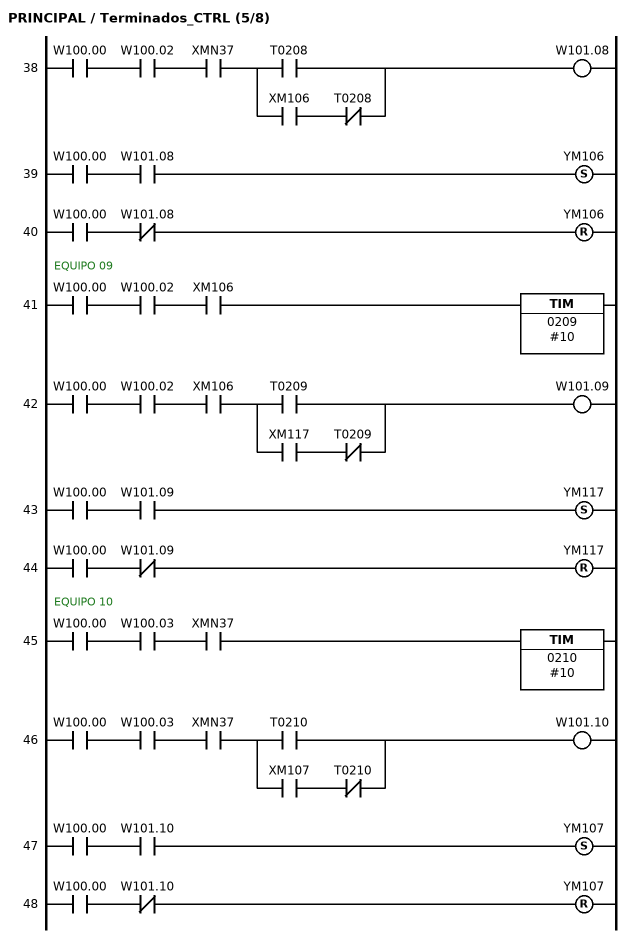
; [picture p24: PRINCIPAL / Terminados_CTRL, rungs 38-48]
; rung 38
LD W100.00
AND W100.02
AND XMN37
LD T0208
LD XM106
ANDNOT T0208
ORLD
ANDLD
OUT W101.08
; rung 39
LD W100.00
AND W101.08
SET YM106
; rung 40
LD W100.00
ANDNOT W101.08
RSET YM106
; rung 41: EQUIPO 09
LD W100.00
AND W100.02
AND XM106
TIM 0209 #10
; rung 42
LD W100.00
AND W100.02
AND XM106
LD T0209
LD XM117
ANDNOT T0209
ORLD
ANDLD
OUT W101.09
; rung 43
LD W100.00
AND W101.09
SET YM117
; rung 44
LD W100.00
ANDNOT W101.09
RSET YM117
; rung 45: EQUIPO 10
LD W100.00
AND W100.03
AND XMN37
TIM 0210 #10
; rung 46
LD W100.00
AND W100.03
AND XMN37
LD T0210
LD XM107
ANDNOT T0210
ORLD
ANDLD
OUT W101.10
; rung 47
LD W100.00
AND W101.10
SET YM107
; rung 48
LD W100.00
ANDNOT W101.10
RSET YM107

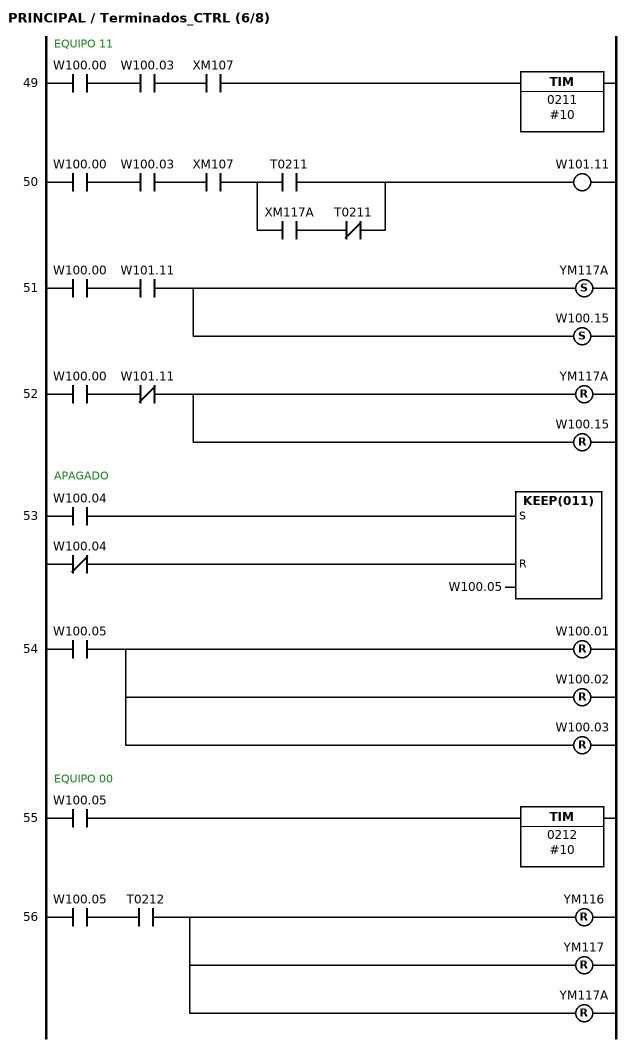
; rung 49: EQUIPO 11
LD W100.00
AND W100.03
AND XM107
TIM 0211 #10
; rung 50
LD W100.00
AND W100.03
AND XM107
LD T0211
LD XM117A
ANDNOT T0211
ORLD
ANDLD
OUT W101.11
; rung 51
LD W100.00
AND W101.11
SET YM117A
SET W100.15
; rung 52
LD W100.00
ANDNOT W101.11
RSET YM117A
RSET W100.15
; rung 53: APAGADO
LD W100.04
LDNOT W100.04
KEEP(011) W100.05
; rung 54
LD W100.05
RSET W100.01
RSET W100.02
RSET W100.03
; rung 55: EQUIPO 00
LD W100.05
TIM 0212 #10
; rung 56
LD W100.05
AND T0212
RSET YM116
RSET YM117
RSET YM117A

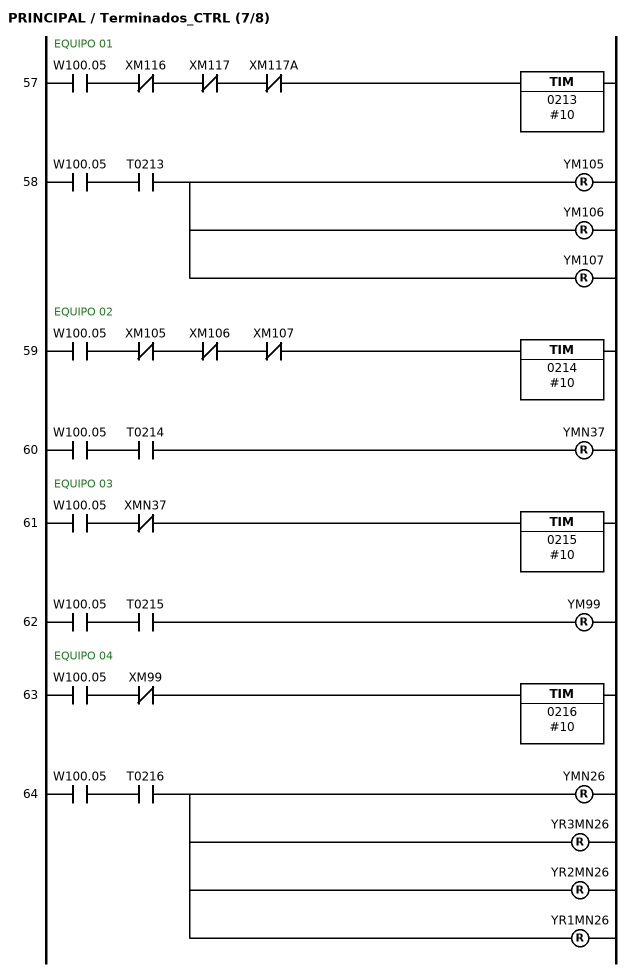
; rung 57: EQUIPO 01
LD W100.05
ANDNOT XM116
ANDNOT XM117
ANDNOT XM117A
TIM 0213 #10
; rung 58
LD W100.05
AND T0213
RSET YM105
RSET YM106
RSET YM107
; rung 59: EQUIPO 02
LD W100.05
ANDNOT XM105
ANDNOT XM106
ANDNOT XM107
TIM 0214 #10
; rung 60
LD W100.05
AND T0214
RSET YMN37
; rung 61: EQUIPO 03
LD W100.05
ANDNOT XMN37
TIM 0215 #10
; rung 62
LD W100.05
AND T0215
RSET YM99
; rung 63: EQUIPO 04
LD W100.05
ANDNOT XM99
TIM 0216 #10
; rung 64
LD W100.05
AND T0216
RSET YMN26
RSET YR3MN26
RSET YR2MN26
RSET YR1MN26

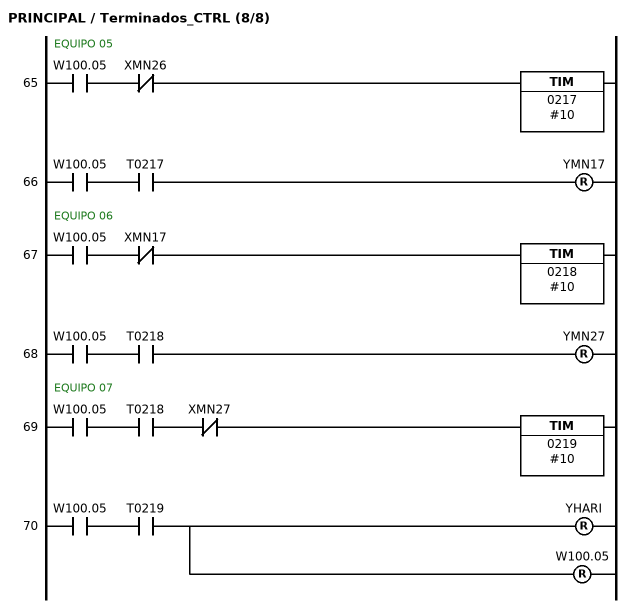
; rung 65: EQUIPO 05
LD W100.05
ANDNOT XMN26
TIM 0217 #10
; rung 66
LD W100.05
AND T0217
RSET YMN17
; rung 67: EQUIPO 06
LD W100.05
ANDNOT XMN17
TIM 0218 #10
; rung 68
LD W100.05
AND T0218
RSET YMN27
; rung 69: EQUIPO 07
LD W100.05
AND T0218
ANDNOT XMN27
TIM 0219 #10
; rung 70
LD W100.05
AND T0219
RSET YHARI
RSET W100.05

### Section Terminados_OUT

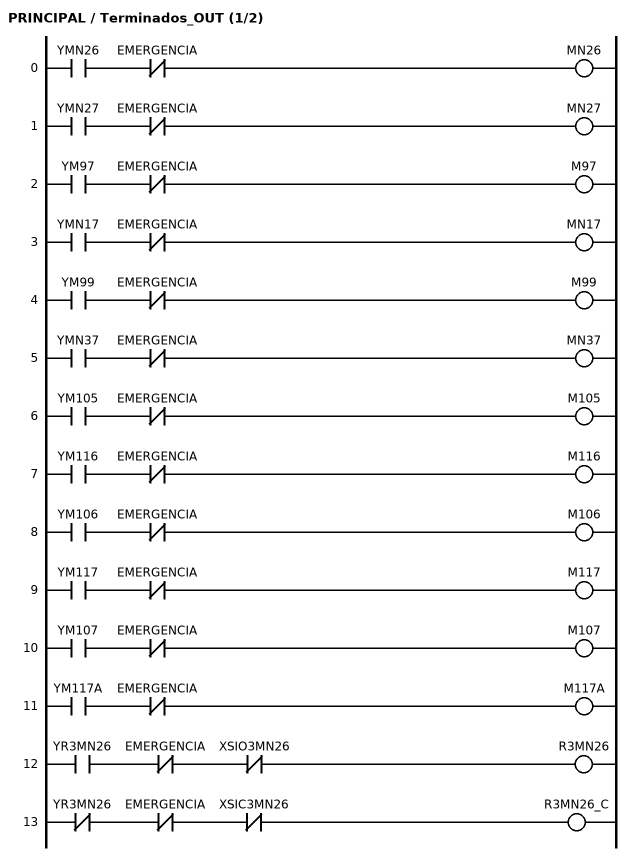
; rung 0
LD YMN26
ANDNOT EMERGENCIA
OUT MN26
; rung 1
LD YMN27
ANDNOT EMERGENCIA
OUT MN27
; rung 2
LD YM97
ANDNOT EMERGENCIA
OUT M97
; rung 3
LD YMN17
ANDNOT EMERGENCIA
OUT MN17
; rung 4
LD YM99
ANDNOT EMERGENCIA
OUT M99
; rung 5
LD YMN37
ANDNOT EMERGENCIA
OUT MN37
; rung 6
LD YM105
ANDNOT EMERGENCIA
OUT M105
; rung 7
LD YM116
ANDNOT EMERGENCIA
OUT M116
; rung 8
LD YM106
ANDNOT EMERGENCIA
OUT M106
; rung 9
LD YM117
ANDNOT EMERGENCIA
OUT M117
; rung 10
LD YM107
ANDNOT EMERGENCIA
OUT M107
; rung 11
LD YM117A
ANDNOT EMERGENCIA
OUT M117A
; rung 12
LD YR3MN26
ANDNOT EMERGENCIA
ANDNOT XSIO3MN26
OUT R3MN26
; rung 13
LDNOT YR3MN26
ANDNOT EMERGENCIA
ANDNOT XSIC3MN26
OUT R3MN26_C

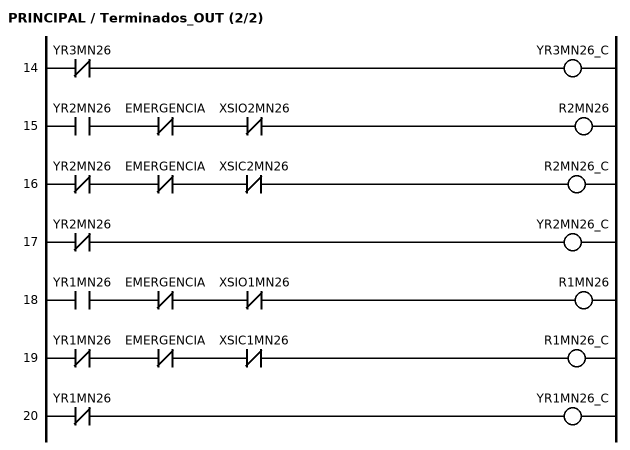
; rung 14
LDNOT YR3MN26
OUT YR3MN26_C
; rung 15
LD YR2MN26
ANDNOT EMERGENCIA
ANDNOT XSIO2MN26
OUT R2MN26
; rung 16
LDNOT YR2MN26
ANDNOT EMERGENCIA
ANDNOT XSIC2MN26
OUT R2MN26_C
; rung 17
LDNOT YR2MN26
OUT YR2MN26_C
; rung 18
LD YR1MN26
ANDNOT EMERGENCIA
ANDNOT XSIO1MN26
OUT R1MN26
; rung 19
LDNOT YR1MN26
ANDNOT EMERGENCIA
ANDNOT XSIC1MN26
OUT R1MN26_C
; rung 20
LDNOT YR1MN26
OUT YR1MN26_C

### Section LPZ_T1_v1_CTRL

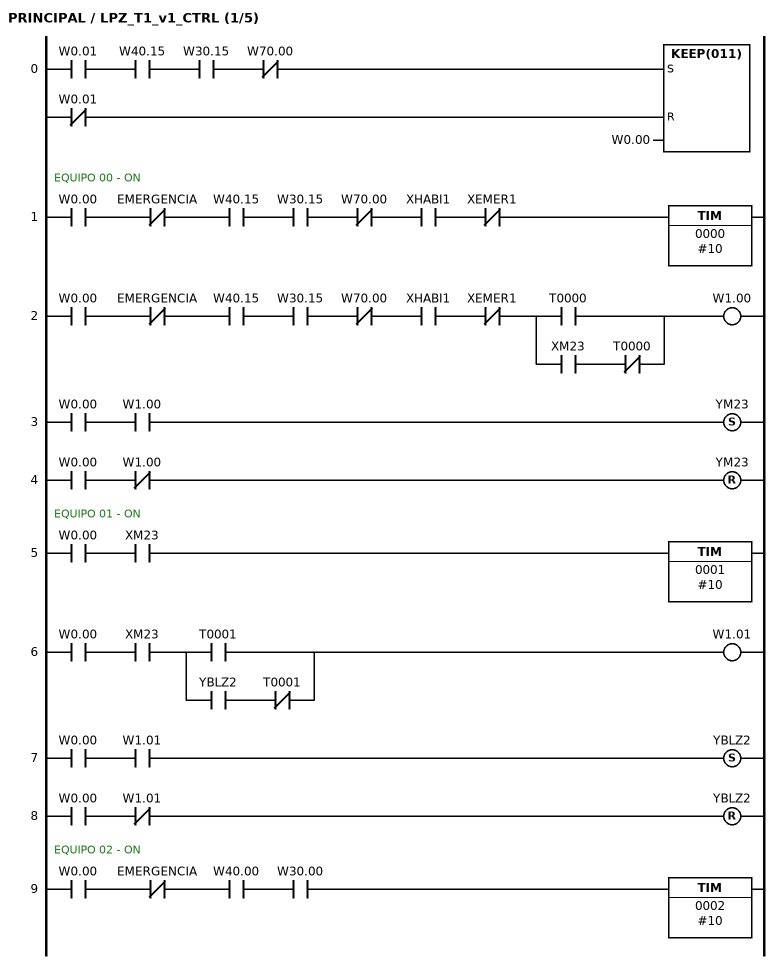
; rung 0
LD W0.01
AND W40.15
AND W30.15
ANDNOT W70.00
LDNOT W0.01
KEEP(011) W0.00
; rung 1: EQUIPO 00 - ON
LD W0.00
ANDNOT EMERGENCIA
AND W40.15
AND W30.15
ANDNOT W70.00
AND XHABI1
ANDNOT XEMER1
TIM 0000 #10
; rung 2
LD W0.00
ANDNOT EMERGENCIA
AND W40.15
AND W30.15
ANDNOT W70.00
AND XHABI1
ANDNOT XEMER1
LD T0000
LD XM23
ANDNOT T0000
ORLD
ANDLD
OUT W1.00
; rung 3
LD W0.00
AND W1.00
SET YM23
; rung 4
LD W0.00
ANDNOT W1.00
RSET YM23
; rung 5: EQUIPO 01 - ON
LD W0.00
AND XM23
TIM 0001 #10
; rung 6
LD W0.00
AND XM23
LD T0001
LD YBLZ2
ANDNOT T0001
ORLD
ANDLD
OUT W1.01
; rung 7
LD W0.00
AND W1.01
SET YBLZ2
; rung 8
LD W0.00
ANDNOT W1.01
RSET YBLZ2
; rung 9: EQUIPO 02 - ON
LD W0.00
ANDNOT EMERGENCIA
AND W40.00
AND W30.00
TIM 0002 #10

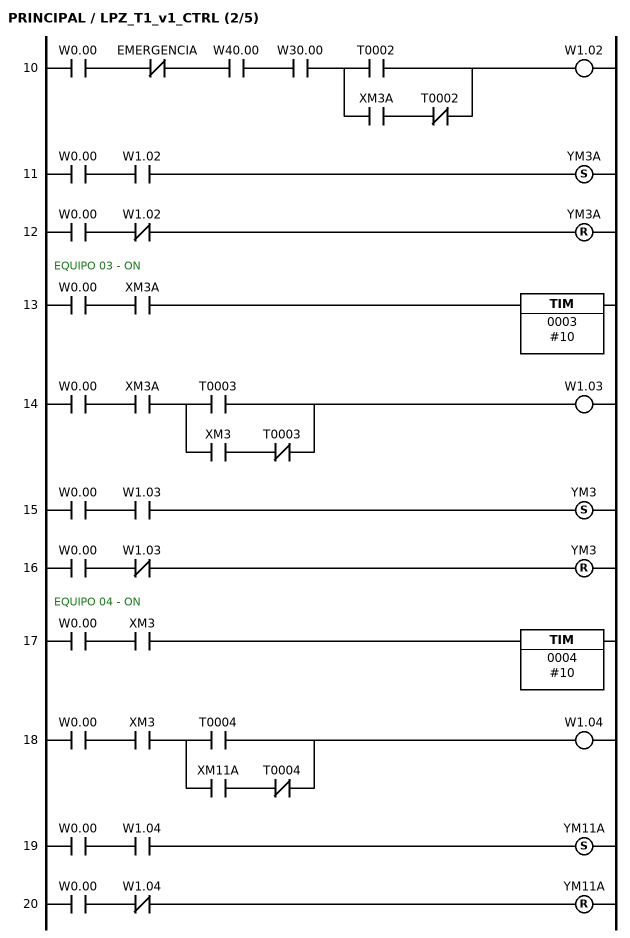
; rung 10
LD W0.00
ANDNOT EMERGENCIA
AND W40.00
AND W30.00
LD T0002
LD XM3A
ANDNOT T0002
ORLD
ANDLD
OUT W1.02
; rung 11
LD W0.00
AND W1.02
SET YM3A
; rung 12
LD W0.00
ANDNOT W1.02
RSET YM3A
; rung 13: EQUIPO 03 - ON
LD W0.00
AND XM3A
TIM 0003 #10
; rung 14
LD W0.00
AND XM3A
LD T0003
LD XM3
ANDNOT T0003
ORLD
ANDLD
OUT W1.03
; rung 15
LD W0.00
AND W1.03
SET YM3
; rung 16
LD W0.00
ANDNOT W1.03
RSET YM3
; rung 17: EQUIPO 04 - ON
LD W0.00
AND XM3
TIM 0004 #10
; rung 18
LD W0.00
AND XM3
LD T0004
LD XM11A
ANDNOT T0004
ORLD
ANDLD
OUT W1.04
; rung 19
LD W0.00
AND W1.04
SET YM11A
; rung 20
LD W0.00
ANDNOT W1.04
RSET YM11A

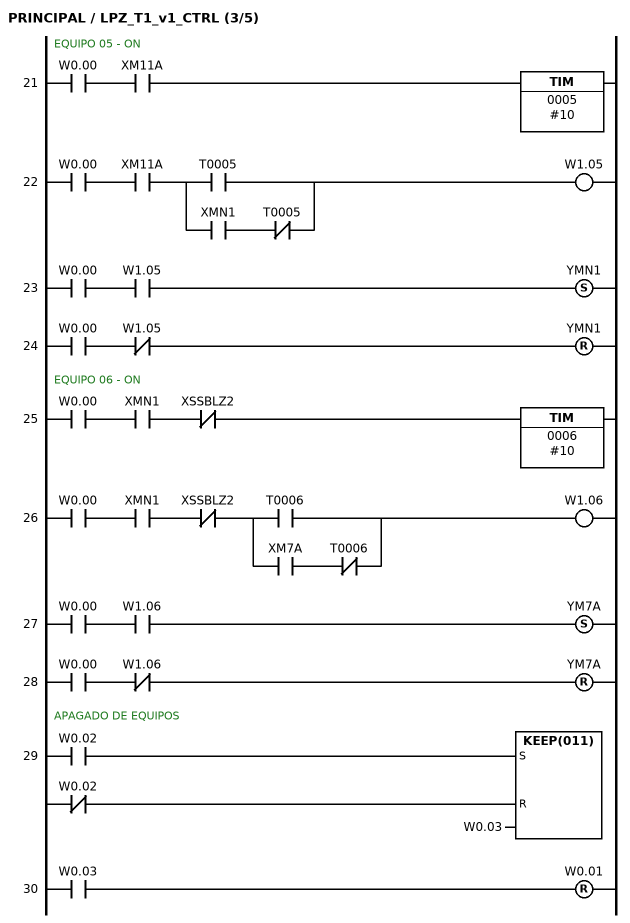
; rung 21: EQUIPO 05 - ON
LD W0.00
AND XM11A
TIM 0005 #10
; rung 22
LD W0.00
AND XM11A
LD T0005
LD XMN1
ANDNOT T0005
ORLD
ANDLD
OUT W1.05
; rung 23
LD W0.00
AND W1.05
SET YMN1
; rung 24
LD W0.00
ANDNOT W1.05
RSET YMN1
; rung 25: EQUIPO 06 - ON
LD W0.00
AND XMN1
ANDNOT XSSBLZ2
TIM 0006 #10
; rung 26
LD W0.00
AND XMN1
ANDNOT XSSBLZ2
LD T0006
LD XM7A
ANDNOT T0006
ORLD
ANDLD
OUT W1.06
; rung 27
LD W0.00
AND W1.06
SET YM7A
; rung 28
LD W0.00
ANDNOT W1.06
RSET YM7A
; rung 29: APAGADO DE EQUIPOS
LD W0.02
LDNOT W0.02
KEEP(011) W0.03
; rung 30
LD W0.03
RSET W0.01

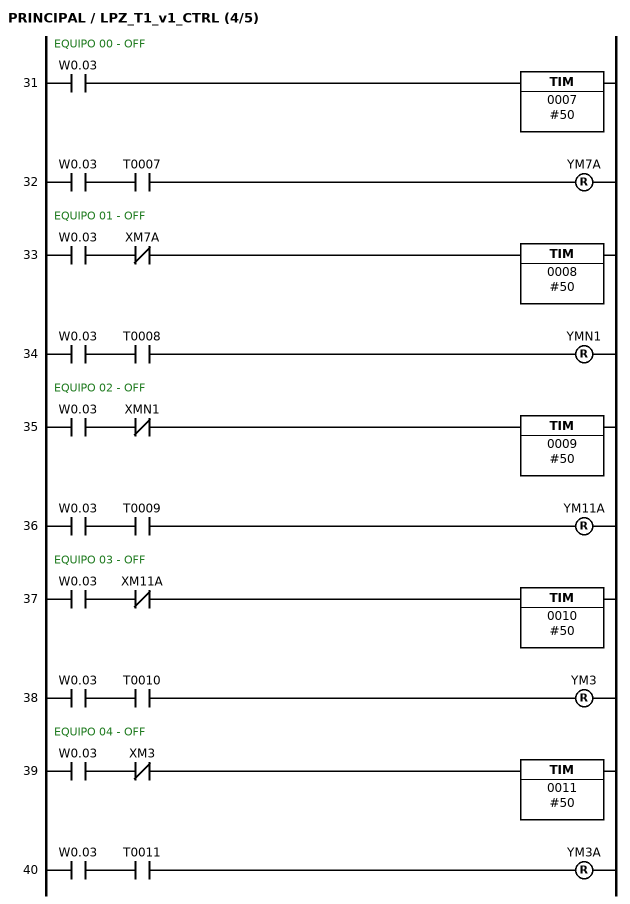
; rung 31: EQUIPO 00 - OFF
LD W0.03
TIM 0007 #50
; rung 32
LD W0.03
AND T0007
RSET YM7A
; rung 33: EQUIPO 01 - OFF
LD W0.03
ANDNOT XM7A
TIM 0008 #50
; rung 34
LD W0.03
AND T0008
RSET YMN1
; rung 35: EQUIPO 02 - OFF
LD W0.03
ANDNOT XMN1
TIM 0009 #50
; rung 36
LD W0.03
AND T0009
RSET YM11A
; rung 37: EQUIPO 03 - OFF
LD W0.03
ANDNOT XM11A
TIM 0010 #50
; rung 38
LD W0.03
AND T0010
RSET YM3
; rung 39: EQUIPO 04 - OFF
LD W0.03
ANDNOT XM3
TIM 0011 #50
; rung 40
LD W0.03
AND T0011
RSET YM3A

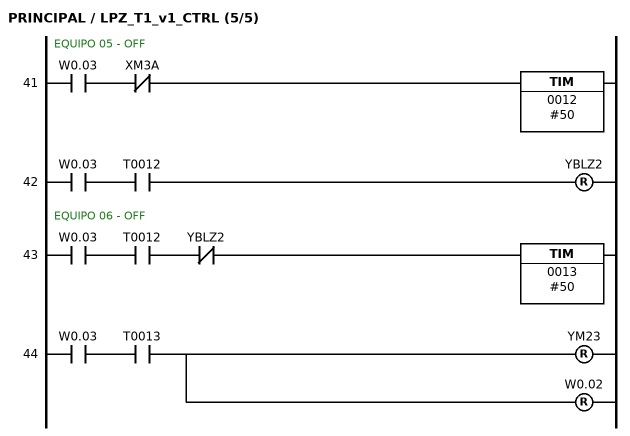
; rung 41: EQUIPO 05 - OFF
LD W0.03
ANDNOT XM3A
TIM 0012 #50
; rung 42
LD W0.03
AND T0012
RSET YBLZ2
; rung 43: EQUIPO 06 - OFF
LD W0.03
AND T0012
ANDNOT YBLZ2
TIM 0013 #50
; rung 44
LD W0.03
AND T0013
RSET YM23
RSET W0.02

### Section LPZ_T1_v2_CTRL

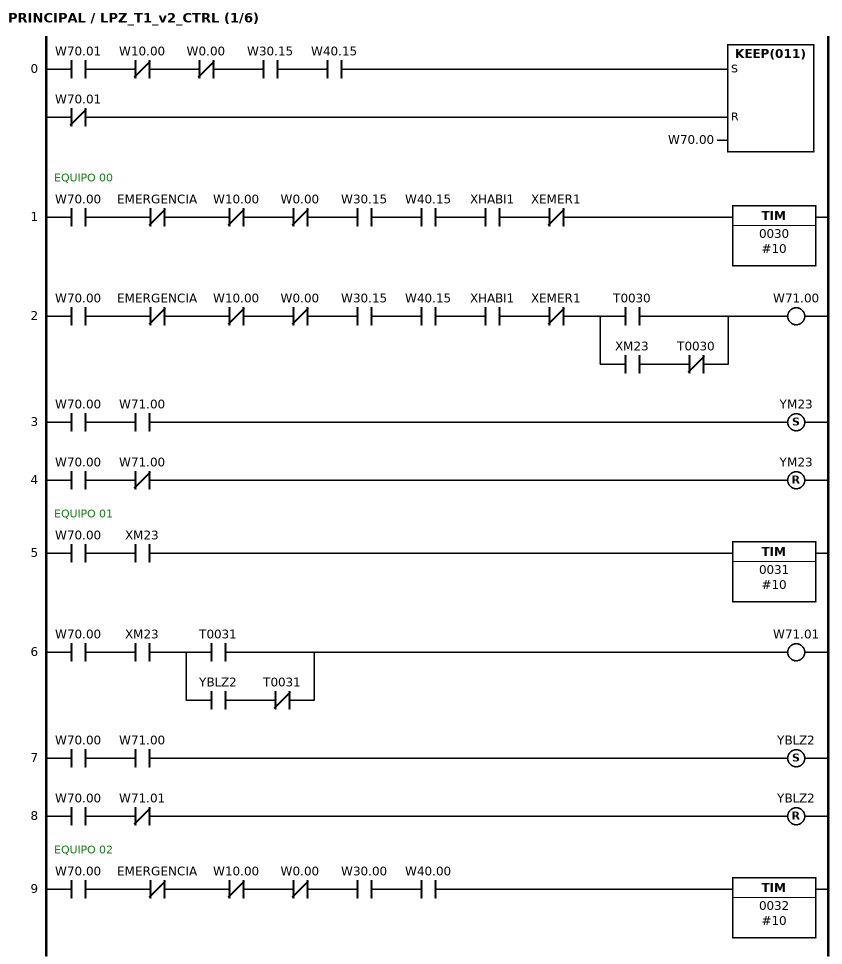
; rung 0
LD W70.01
ANDNOT W10.00
ANDNOT W0.00
AND W30.15
AND W40.15
LDNOT W70.01
KEEP(011) W70.00
; rung 1: EQUIPO 00
LD W70.00
ANDNOT EMERGENCIA
ANDNOT W10.00
ANDNOT W0.00
AND W30.15
AND W40.15
AND XHABI1
ANDNOT XEMER1
TIM 0030 #10
; rung 2
LD W70.00
ANDNOT EMERGENCIA
ANDNOT W10.00
ANDNOT W0.00
AND W30.15
AND W40.15
AND XHABI1
ANDNOT XEMER1
LD T0030
LD XM23
ANDNOT T0030
ORLD
ANDLD
OUT W71.00
; rung 3
LD W70.00
AND W71.00
SET YM23
; rung 4
LD W70.00
ANDNOT W71.00
RSET YM23
; rung 5: EQUIPO 01
LD W70.00
AND XM23
TIM 0031 #10
; rung 6
LD W70.00
AND XM23
LD T0031
LD YBLZ2
ANDNOT T0031
ORLD
ANDLD
OUT W71.01
; rung 7
LD W70.00
AND W71.00
SET YBLZ2
; rung 8
LD W70.00
ANDNOT W71.01
RSET YBLZ2
; rung 9: EQUIPO 02
LD W70.00
ANDNOT EMERGENCIA
ANDNOT W10.00
ANDNOT W0.00
AND W30.00
AND W40.00
TIM 0032 #10

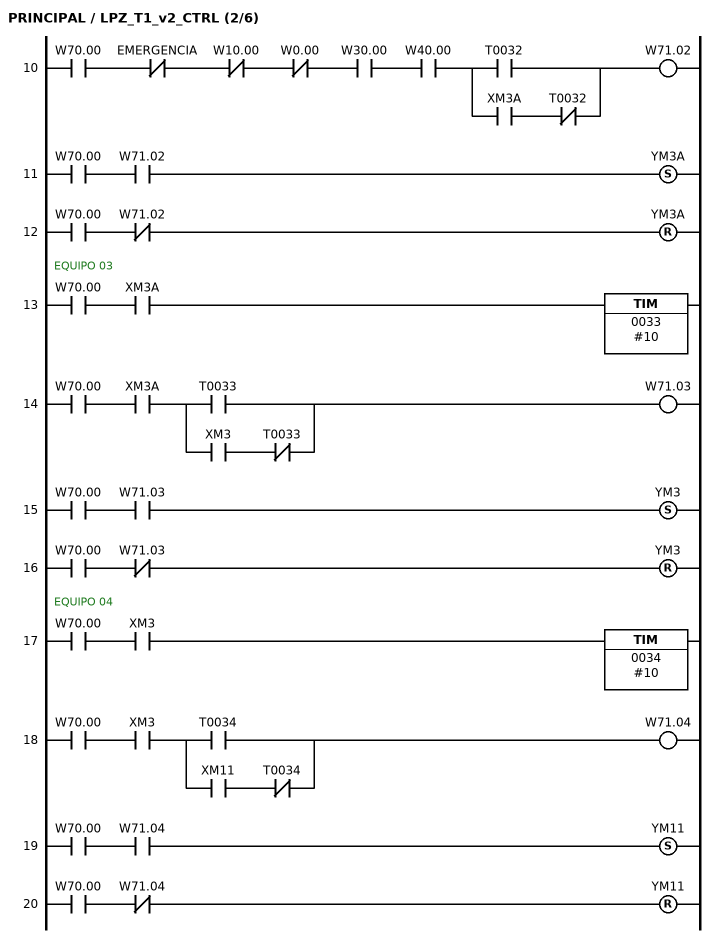
; rung 10
LD W70.00
ANDNOT EMERGENCIA
ANDNOT W10.00
ANDNOT W0.00
AND W30.00
AND W40.00
LD T0032
LD XM3A
ANDNOT T0032
ORLD
ANDLD
OUT W71.02
; rung 11
LD W70.00
AND W71.02
SET YM3A
; rung 12
LD W70.00
ANDNOT W71.02
RSET YM3A
; rung 13: EQUIPO 03
LD W70.00
AND XM3A
TIM 0033 #10
; rung 14
LD W70.00
AND XM3A
LD T0033
LD XM3
ANDNOT T0033
ORLD
ANDLD
OUT W71.03
; rung 15
LD W70.00
AND W71.03
SET YM3
; rung 16
LD W70.00
ANDNOT W71.03
RSET YM3
; rung 17: EQUIPO 04
LD W70.00
AND XM3
TIM 0034 #10
; rung 18
LD W70.00
AND XM3
LD T0034
LD XM11
ANDNOT T0034
ORLD
ANDLD
OUT W71.04
; rung 19
LD W70.00
AND W71.04
SET YM11
; rung 20
LD W70.00
ANDNOT W71.04
RSET YM11

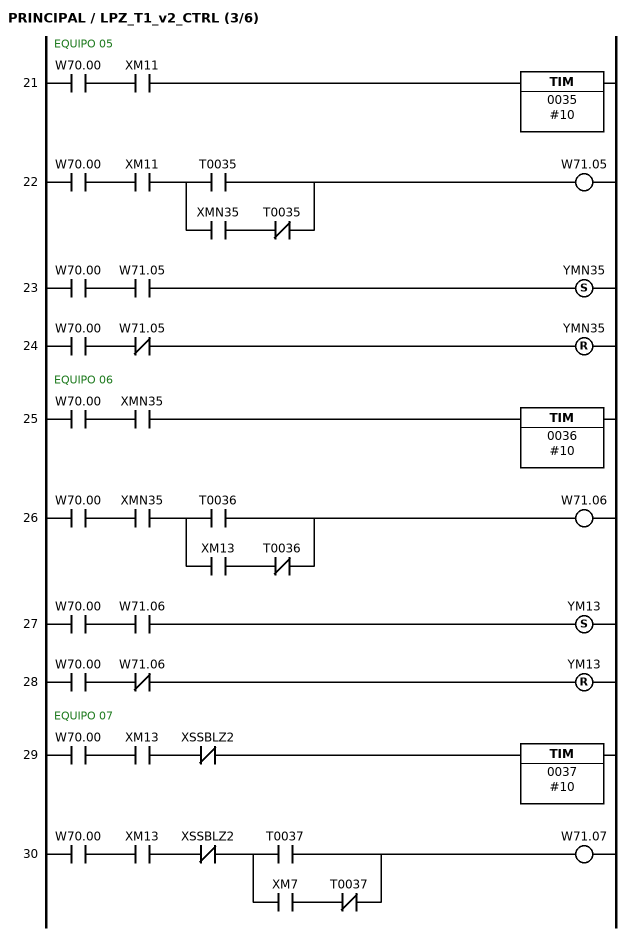
; rung 21: EQUIPO 05
LD W70.00
AND XM11
TIM 0035 #10
; rung 22
LD W70.00
AND XM11
LD T0035
LD XMN35
ANDNOT T0035
ORLD
ANDLD
OUT W71.05
; rung 23
LD W70.00
AND W71.05
SET YMN35
; rung 24
LD W70.00
ANDNOT W71.05
RSET YMN35
; rung 25: EQUIPO 06
LD W70.00
AND XMN35
TIM 0036 #10
; rung 26
LD W70.00
AND XMN35
LD T0036
LD XM13
ANDNOT T0036
ORLD
ANDLD
OUT W71.06
; rung 27
LD W70.00
AND W71.06
SET YM13
; rung 28
LD W70.00
ANDNOT W71.06
RSET YM13
; rung 29: EQUIPO 07
LD W70.00
AND XM13
ANDNOT XSSBLZ2
TIM 0037 #10
; rung 30
LD W70.00
AND XM13
ANDNOT XSSBLZ2
LD T0037
LD XM7
ANDNOT T0037
ORLD
ANDLD
OUT W71.07

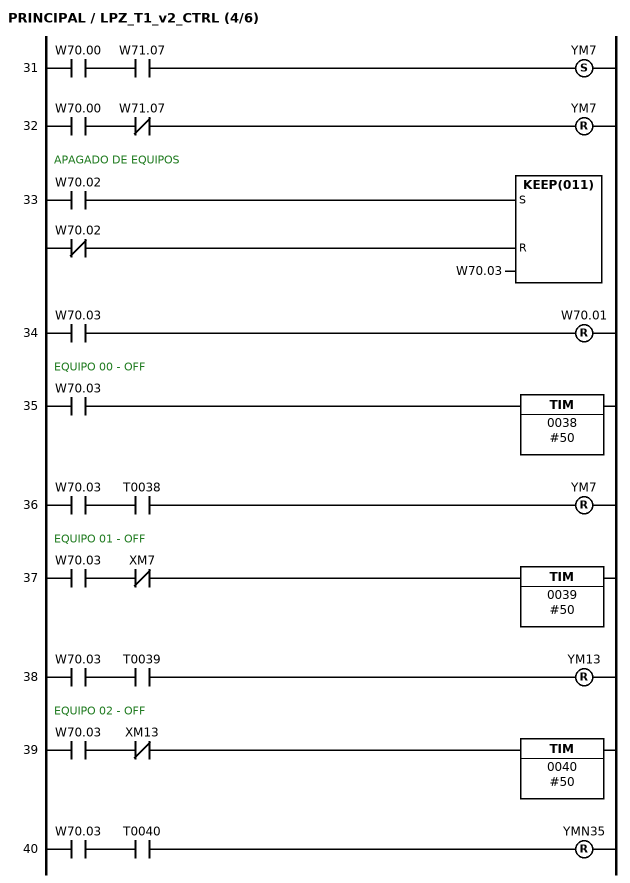
; rung 31
LD W70.00
AND W71.07
SET YM7
; rung 32
LD W70.00
ANDNOT W71.07
RSET YM7
; rung 33: APAGADO DE EQUIPOS
LD W70.02
LDNOT W70.02
KEEP(011) W70.03
; rung 34
LD W70.03
RSET W70.01
; rung 35: EQUIPO 00 - OFF
LD W70.03
TIM 0038 #50
; rung 36
LD W70.03
AND T0038
RSET YM7
; rung 37: EQUIPO 01 - OFF
LD W70.03
ANDNOT XM7
TIM 0039 #50
; rung 38
LD W70.03
AND T0039
RSET YM13
; rung 39: EQUIPO 02 - OFF
LD W70.03
ANDNOT XM13
TIM 0040 #50
; rung 40
LD W70.03
AND T0040
RSET YMN35

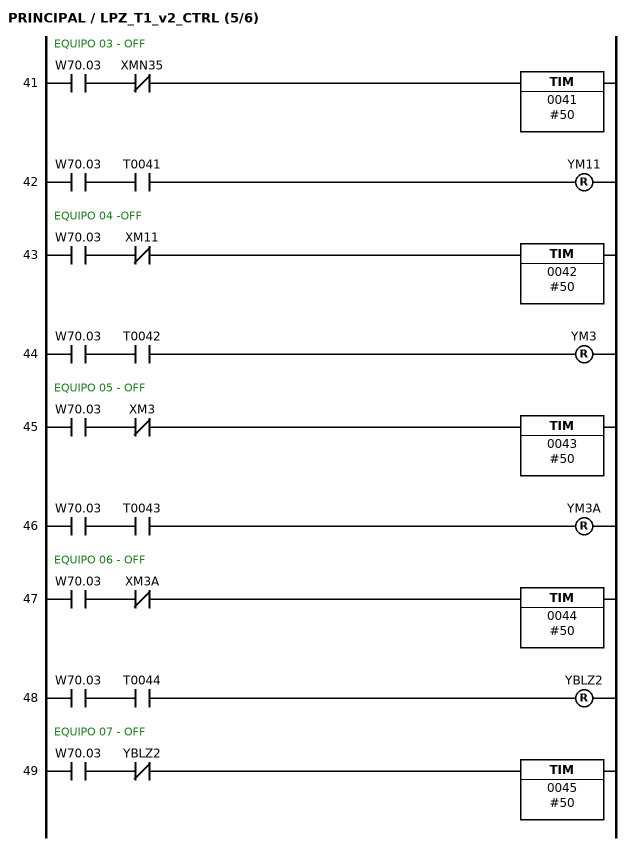
; rung 41: EQUIPO 03 - OFF
LD W70.03
ANDNOT XMN35
TIM 0041 #50
; rung 42
LD W70.03
AND T0041
RSET YM11
; rung 43: EQUIPO 04 -OFF
LD W70.03
ANDNOT XM11
TIM 0042 #50
; rung 44
LD W70.03
AND T0042
RSET YM3
; rung 45: EQUIPO 05 - OFF
LD W70.03
ANDNOT XM3
TIM 0043 #50
; rung 46
LD W70.03
AND T0043
RSET YM3A
; rung 47: EQUIPO 06 - OFF
LD W70.03
ANDNOT XM3A
TIM 0044 #50
; rung 48
LD W70.03
AND T0044
RSET YBLZ2
; rung 49: EQUIPO 07 - OFF
LD W70.03
ANDNOT YBLZ2
TIM 0045 #50

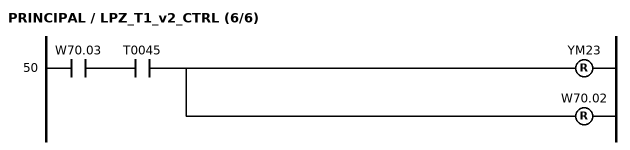
; rung 50
LD W70.03
AND T0045
RSET YM23
RSET W70.02

### Section LPZ_T1_OUT

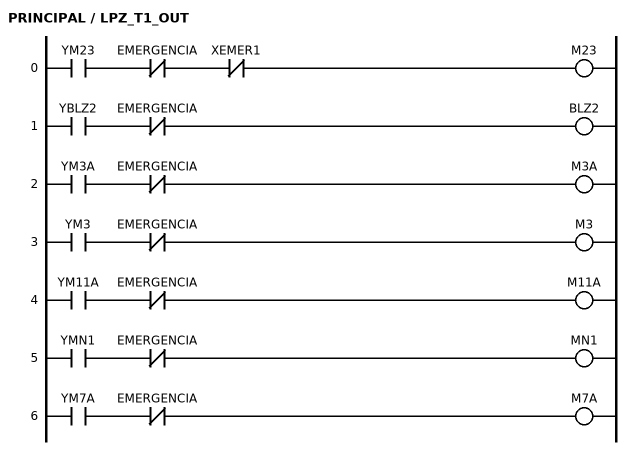
; rung 0
LD YM23
ANDNOT EMERGENCIA
ANDNOT XEMER1
OUT M23
; rung 1
LD YBLZ2
ANDNOT EMERGENCIA
OUT BLZ2
; rung 2
LD YM3A
ANDNOT EMERGENCIA
OUT M3A
; rung 3
LD YM3
ANDNOT EMERGENCIA
OUT M3
; rung 4
LD YM11A
ANDNOT EMERGENCIA
OUT M11A
; rung 5
LD YMN1
ANDNOT EMERGENCIA
OUT MN1
; rung 6
LD YM7A
ANDNOT EMERGENCIA
OUT M7A

### Section LPZ_2Rociado_CTRL

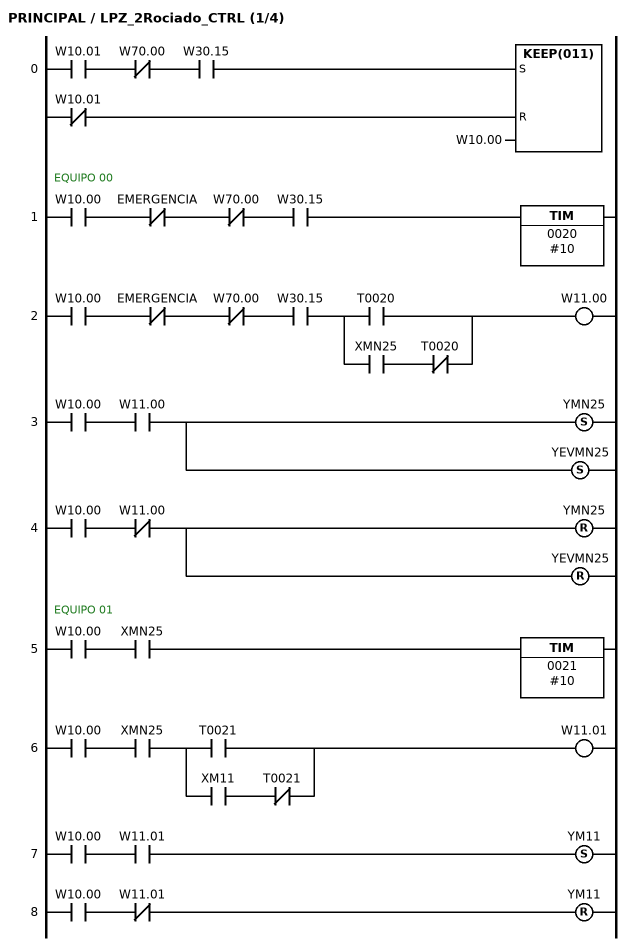
; rung 0
LD W10.01
ANDNOT W70.00
AND W30.15
LDNOT W10.01
KEEP(011) W10.00
; rung 1: EQUIPO 00
LD W10.00
ANDNOT EMERGENCIA
ANDNOT W70.00
AND W30.15
TIM 0020 #10
; rung 2
LD W10.00
ANDNOT EMERGENCIA
ANDNOT W70.00
AND W30.15
LD T0020
LD XMN25
ANDNOT T0020
ORLD
ANDLD
OUT W11.00
; rung 3
LD W10.00
AND W11.00
SET YMN25
SET YEVMN25
; rung 4
LD W10.00
ANDNOT W11.00
RSET YMN25
RSET YEVMN25
; rung 5: EQUIPO 01
LD W10.00
AND XMN25
TIM 0021 #10
; rung 6
LD W10.00
AND XMN25
LD T0021
LD XM11
ANDNOT T0021
ORLD
ANDLD
OUT W11.01
; rung 7
LD W10.00
AND W11.01
SET YM11
; rung 8
LD W10.00
ANDNOT W11.01
RSET YM11

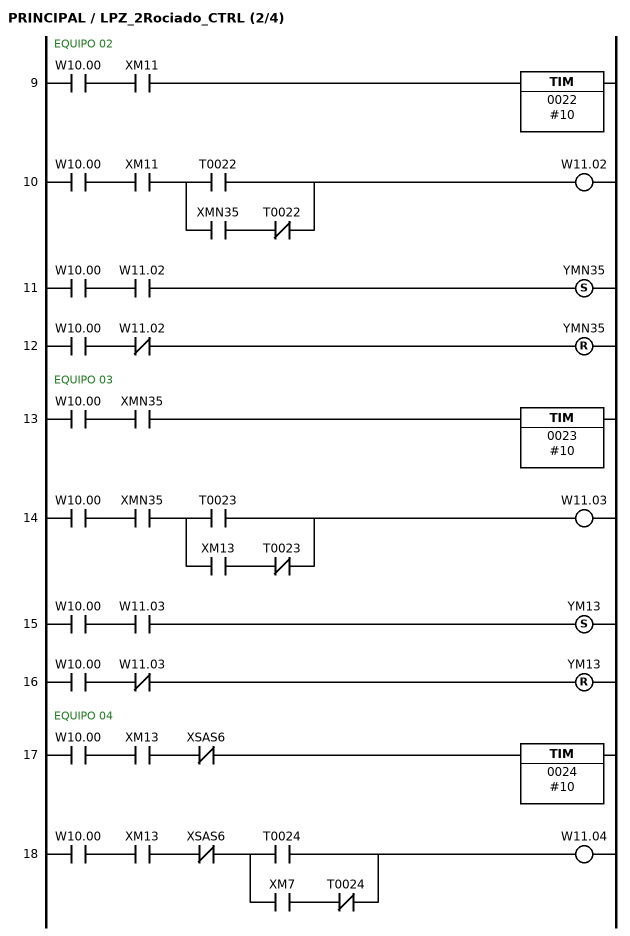
; rung 9: EQUIPO 02
LD W10.00
AND XM11
TIM 0022 #10
; rung 10
LD W10.00
AND XM11
LD T0022
LD XMN35
ANDNOT T0022
ORLD
ANDLD
OUT W11.02
; rung 11
LD W10.00
AND W11.02
SET YMN35
; rung 12
LD W10.00
ANDNOT W11.02
RSET YMN35
; rung 13: EQUIPO 03
LD W10.00
AND XMN35
TIM 0023 #10
; rung 14
LD W10.00
AND XMN35
LD T0023
LD XM13
ANDNOT T0023
ORLD
ANDLD
OUT W11.03
; rung 15
LD W10.00
AND W11.03
SET YM13
; rung 16
LD W10.00
ANDNOT W11.03
RSET YM13
; rung 17: EQUIPO 04
LD W10.00
AND XM13
ANDNOT XSAS6
TIM 0024 #10
; rung 18
LD W10.00
AND XM13
ANDNOT XSAS6
LD T0024
LD XM7
ANDNOT T0024
ORLD
ANDLD
OUT W11.04

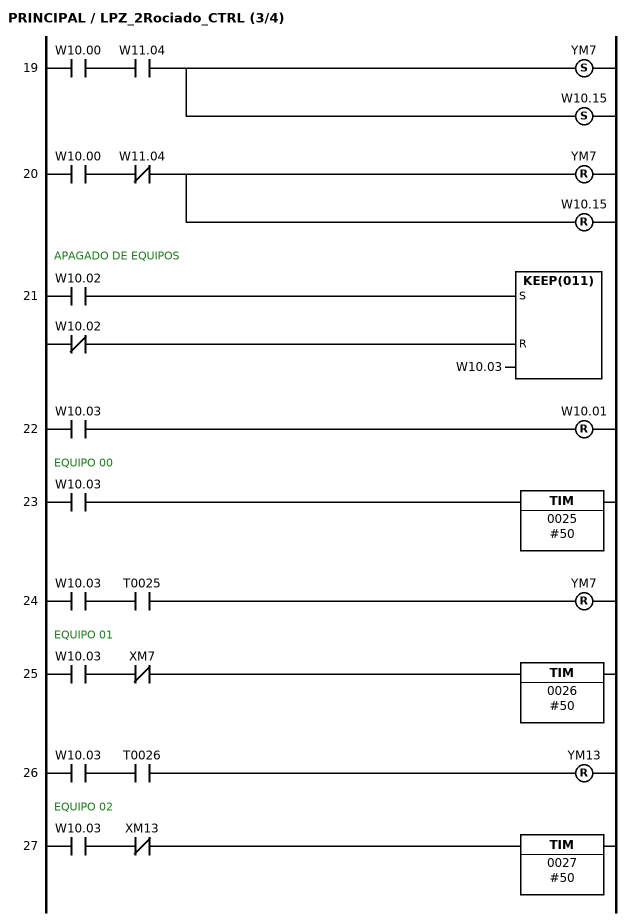
; rung 19
LD W10.00
AND W11.04
SET YM7
SET W10.15
; rung 20
LD W10.00
ANDNOT W11.04
RSET YM7
RSET W10.15
; rung 21: APAGADO DE EQUIPOS
LD W10.02
LDNOT W10.02
KEEP(011) W10.03
; rung 22
LD W10.03
RSET W10.01
; rung 23: EQUIPO 00
LD W10.03
TIM 0025 #50
; rung 24
LD W10.03
AND T0025
RSET YM7
; rung 25: EQUIPO 01
LD W10.03
ANDNOT XM7
TIM 0026 #50
; rung 26
LD W10.03
AND T0026
RSET YM13
; rung 27: EQUIPO 02
LD W10.03
ANDNOT XM13
TIM 0027 #50

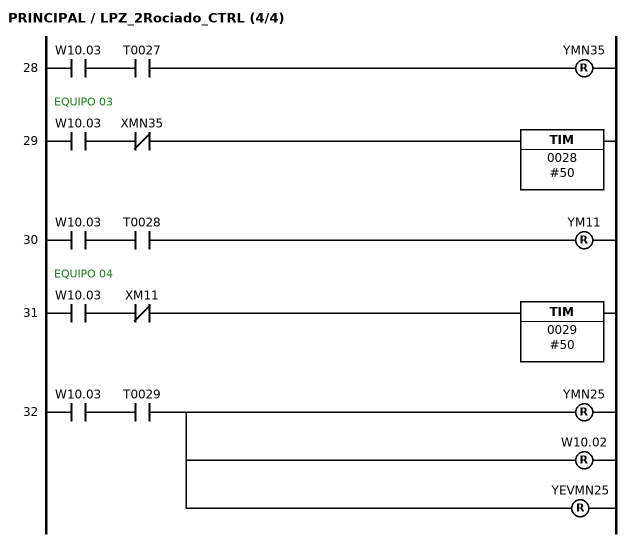
; rung 28
LD W10.03
AND T0027
RSET YMN35
; rung 29: EQUIPO 03
LD W10.03
ANDNOT XMN35
TIM 0028 #50
; rung 30
LD W10.03
AND T0028
RSET YM11
; rung 31: EQUIPO 04
LD W10.03
ANDNOT XM11
TIM 0029 #50
; rung 32
LD W10.03
AND T0029
RSET YMN25
RSET W10.02
RSET YEVMN25

### Section LPZ_2Rociado_OUT

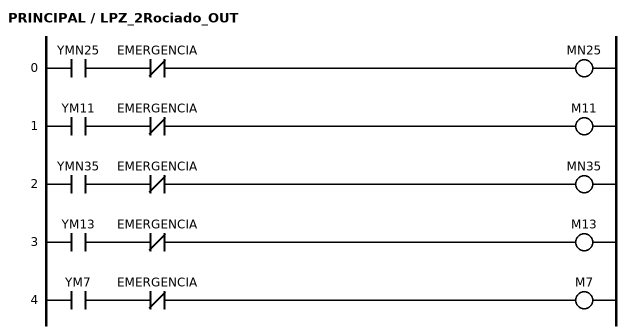
; rung 0
LD YMN25
ANDNOT EMERGENCIA
OUT MN25
; rung 1
LD YM11
ANDNOT EMERGENCIA
OUT M11
; rung 2
LD YMN35
ANDNOT EMERGENCIA
OUT MN35
; rung 3
LD YM13
ANDNOT EMERGENCIA
OUT M13
; rung 4
LD YM7
ANDNOT EMERGENCIA
OUT M7

### Section LPZ_Residuos_CTRL

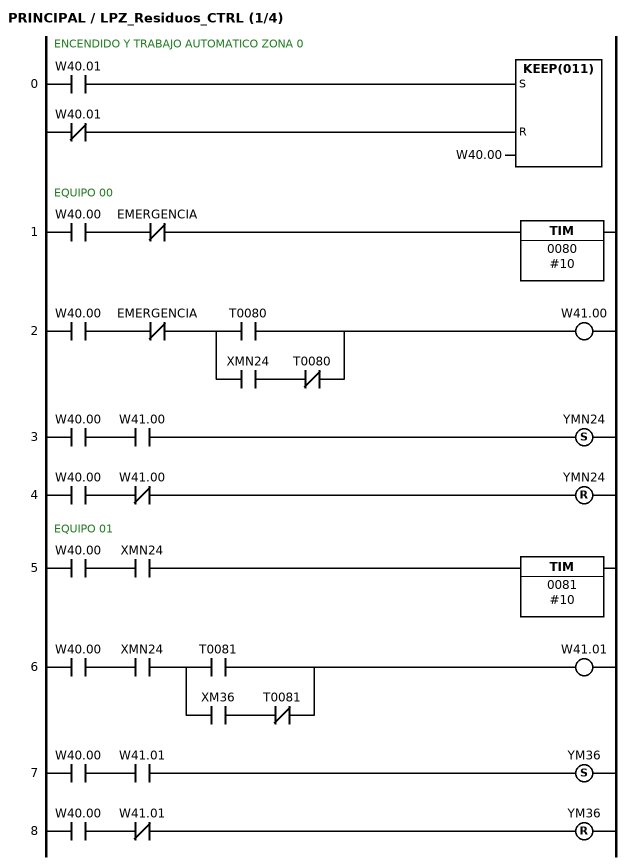
; rung 0: ENCENDIDO Y TRABAJO AUTOMATICO ZONA 0
LD W40.01
LDNOT W40.01
KEEP(011) W40.00
; rung 1: EQUIPO 00
LD W40.00
ANDNOT EMERGENCIA
TIM 0080 #10
; rung 2
LD W40.00
ANDNOT EMERGENCIA
LD T0080
LD XMN24
ANDNOT T0080
ORLD
ANDLD
OUT W41.00
; rung 3
LD W40.00
AND W41.00
SET YMN24
; rung 4
LD W40.00
ANDNOT W41.00
RSET YMN24
; rung 5: EQUIPO 01
LD W40.00
AND XMN24
TIM 0081 #10
; rung 6
LD W40.00
AND XMN24
LD T0081
LD XM36
ANDNOT T0081
ORLD
ANDLD
OUT W41.01
; rung 7
LD W40.00
AND W41.01
SET YM36
; rung 8
LD W40.00
ANDNOT W41.01
RSET YM36

